FUNCTION_BLOCK "Test_Function_Block"
{ S7_Optimized_Access := 'TRUE' }
VERSION : 0.1

BEGIN
	// Kan i se det her??
END_FUNCTION_BLOCK

